Staubli VAL3: Apilar.pjx

--- Apilar.pjx ---
Parameters version=s7.10 stackSize=5000 millimeterUnit=true
Program file=_GLOBAL.pgx
Program file=_INFO.pgx
Program file=ajustar.pgx
Program file=getNum.pgx
Program file=inicializar.pgx
Program file=lower.pgx
Program file=mcp.pgx
Program file=putButton.pgx
Program file=putEx.pgx
Program file=putEx2.pgx
Program file=robot.pgx
Program file=robotGet.pgx
Program file=robotPut.pgx
Program file=start.pgx
Program file=stop.pgx
Data file=Apilar.dtx

--- Apilar.dtx ---
bool bTraslada = true
bool bFin
bool bPiezaPreparada
bool bTermina
frame fTrabajo = {x=-400, y=175, z=-274.326706, fatherId=world[0]}
jointRx jHome
public mdesc mNomSpeed = {leave=25, reach=25}
mdesc mVelAprox = {accel=25, vel=50, decel=25, blend=off}
num nPiezaActual = 1
num nTrasladadas = 7
num nPiezaAltura = 12
num nSeparacion = 100
num nTotalPiezas = 2
pointRx p0 = {ry=180, fatherId=fTrabajo[0]}
pointRx pCentro = {x=-400, y=175, z=-272, ry=180, shoulder=righty, elbow=enegative, wrist=wnegative, fatherId=world[0]}
pointRx pDestino = {x=-2.694223E-15, y=50, z=22, rx=-180, ry=7.016709E-15, rz=-180, fatherId=fTrabajo[0]}
pointRx pEntrada = {y=-50, z=103, rx=-180, rz=-180, fatherId=fTrabajo[0]}
pointRx pOrigen = {x=-1.347111E-15, y=-50, z=11, rx=-180, ry=7.016709E-15, rz=-180, fatherId=fTrabajo[0]}
pointRx pEspera = {x=-6.123234E-15, z=50, rx=-180, ry=7.016709E-15, rz=-180, fatherId=fTrabajo[0]}
pointRx pSalida = {x=-1.347111E-15, y=50, z=11, rx=-180, ry=7.016709E-15, rz=-180, fatherId=fTrabajo[0]}
tool tEyector = {z=22, fatherId=flange[0], ioLink=valve1, ioOpen=1, ioClose=1}
trsf trAprox = {z=-50}
num nEspera
num nOffset
bool bHaciaSalida
pointRx pInicio = {fatherId=world[0]}

--- start.pgx ---
program start()
begin
  // Se pone en marcha la aplicacion

  // Se inicializar la aplicacion
  call inicializar()
  call ajustar()

  // Se crean las tareas de la aplicacion
  taskCreate "mcp",100,mcp()
  taskCreate "robot",100,robot()
end

--- _GLOBAL.pgx ---
program _GLOBAL()
begin
  // BOOL
  // - bFin: indicador de finalizacion
  // - bHaciaSalida: indica la direccion del traslado de piezas
  // - bPiezaPreparada: pieza preparada para ser cogida
  // - bTermina: orden de abandonar la ejecucion de la aplicacion
  // - bTraslada: orden de trasladar la pila de piezas
  //
  // FRAME
  // frTrabajo: sistema de coordenadas del area de trabajo
  //
  // JOINT
  // - jHome: brazo en la posicion de referencia
  //
  // MDESC
  // - mNomSpeed: descriptor de movimiento a velocidad nominal
  // - mVelAprox: descriptor de movimiento a velocidad de aproximacion
  //
  // NUM
  // - nEspera: tiempo de espera en la posicion de espera antes de volver a
  //   trasladar la pila de piezas
  // - nOffset: desplazamiento de la posicion de reposo con respecto a la
  //   altura de la pila de piezas.
  // - nPiezaActual: posicion de la proxima pieza a trasladar en la pila origen
  // - nPiezaAltura: altura de la pieza a trasladar
  // - nSeparacion: distancia entre las pilas de bloques
  // - nTotalPiezas: numero total de piezas en la pila
  // - nTrasladadas: numero total acumulado de piezas trasladadas
  //
  // POINT
  // - p0: punto situado en el centro de coordenadas del espacio de trabajo
  // - pCentro: posicion central de referencia del espacio de trabajo
  // - pDestino: posicion de la proxima pieza a colocar
  // - pEntrada: posicion de la pila de entrada
  // - pEspera: posicion de reposo
  // - pInicio: posicion inicial que señala la posicion de la pila de entrada
  // - pOrigen: posicion de la proxima pieza a coger
  // - pSalida: posicion de la pila de salida
  //
  // TOOL
  // - tEyector: parametros de la herramienta (eyector de vacio con ventosas)
  //
  // TRSF
  // - trAprox: transformacion de aproximacion a las posiciones origen/destino
end

--- _INFO.pgx ---
program _INFO()
begin
  // APLILAR (Nivel 2)
  //
  // Traslada indefinidamente una pila de un determinado numero de piezas de
  // una posicion a otra.
  //
  // Version 0.0
  // copyright (c) 2022 victortorreslopez
  // GNU General Public License
  //
  // HISTORIAL DE VERSIONES
  // ----------------------
  // 0.0, 13/12/2022, VTL: creacion (desde PickPlace, 2018)
  //
  // FUNCIONALIDAD
  // -------------
  // - F1: Activa/Desactiva el modo "Trasladar".
  // - F3: Edita el numero total de piezas en la pila a trasladar.
  // - F4: Ajusta el tiempo de espera entre traslados.
  // - F6: Reinicia el contador total de piezas trasladadas.
  // - F8: Sale de la aplicacion.
  //
  // SITUACION INICIAL
  // -----------------
  // - Brazo en su posicion de referencia.
  // - Pila con el numero determinado de bloques en la posicion de entrada.
  // - Ninguna pieza en la posicion de salida.
  // - Antes de ejecutar por primera vez la aplicacion deben ajustarse al valor
  //   deseado las variables: nEspera, nPiezaAltura y nSeparacion.
  //
  // RECURSOS
  // --------
  // - Datos: BOOL, FRAME, JOINT, MDESC, POINT, STRING, TOOL, TRSF.
  // - Instrucciones: appro, title, userPage, while, cls, call, toString, if,
  //   getKey, switch, delay, movej, waitEndMove, for, taskCreate.
  // - Funciones:  getNum, lower, putButton, putEx, putEx2, robotGet, robotPut
  //
  // NOTAS
  // -----
  // - El area de trabajo es una plataforma elevada a 100 mm del suelo.
  // - Pilas de entrada y salida simetricas con respecto al centro del espacio
  //   de trabajo a una distancia "nSeparacion".
  // - En el modo trasladar las piezas se trasladan indefinidamente de la pila
  //   de entrada a la de salida y viceversa.
  // - El espacio de trabajo (fTrabajo) se determina a partir de una posicion
  //   que determina su centro de coordenadas (pCentro)
  //
  // REFERENCIAS
  // -----------
  //
  // CELDA
  // -----
  // - Version: s7.10
  // - Tipo de robot: TX60
  // - Montaje: suelo
  // - Modo usrIn0: directo.
  //
  // DATOS
  // -----
  // - Plataforma = 400x300x3 mm
  // - Altura de la plataforma = 100 mm
  // - Pieza = 69x23x12 mm
  // - Herramienta (eyector) = 40.0x33.3x22.0 mm
end

--- ajustar.pgx ---
program ajustar()
begin
  // Calcula la posiciones de referencia

  // Posicion de entrada y salida
  // - Simetricas con respecto al origen (nSeparacion)
  // - A la altura de la primera pieza
  pEntrada=appro(p0,{0,-nSeparacion/2,-nPiezaAltura,0,0,0})
  pSalida=appro(p0,{0,nSeparacion/2,-nPiezaAltura,0,0,0})

  // Posicion de espera en el centro por encima (offset) de la altura de la pila
  pEspera=appro(p0,{0,0,-((nTotalPiezas*nPiezaAltura)+nOffset),0,0,0})

  // Posicion de espera inicial por encima (offset) de la pila de entrada
  pInicio=appro(pEntrada,{0,0, -((nTotalPiezas*nPiezaAltura)+nOffset),0,0,0})
  end

--- getNum.pgx ---
public program getNum(num nX, num nY, string sFormat, num& nValue)
  local num i
  local num n
  local string s
begin
  // Acquires a number
  //
  // copyright (c) 2013-2021 victortorreslopez
  //
  // GNU General Public License
  //
  // Parameters
  // - nX: cursor column (0 to 39)
  // - nY: cursor row (0 to 13)
  // - sFormat: display format
  // - &nValue: numerical variable to be set
  //
  // Local variables
  // - i: iterator index
  // - n: number of characters in nValue
  // - s: a string
  //
  // Version history
  // ---------------
  // 0.1, 2021/12/30, VTL: 1s update (coding style)
  // 0.0, 2013/12/10, VTL: alfa release

  // Fills s with spaces
  s = ""
  n = len(toString(sFormat, nValue))
  for i = 0 to n - 1
    s = s + " "
  endFor

  // Displays spaces before acquires the new string value
  gotoxy(nX, nY)
  put(s)

  // Acquires the new numerical value
  gotoxy(nX, nY)
  get(nValue)
end

--- inicializar.pgx ---
program inicializar()
begin
  // Pone en marcha la aplicacion

  // Se establece el valor inicial de variables globales
  // BOOL
  bFin=false
  bHaciaSalida=true
  bPiezaPreparada=false
  bTermina=false
  bTraslada=false

  // FRAME
  // Se determina el centro de coordenadas de fTrabajo a partir de la posicion
  // central de referencia de todo el espacio de trabajo (pCentro)
  fTrabajo.trsf.x=pCentro.trsf.x
  fTrabajo.trsf.y=pCentro.trsf.y
  fTrabajo.trsf.z=pCentro.trsf.z

  // NUM
  nOffset=5
  nPiezaActual=0
  nPiezaAltura=12
  nSeparacion=100
  nTotalPiezas=1
  nTrasladadas=0
end

--- lower.pgx ---
public program lower(string& sText)
  local num i
  local num n
begin
  // Converts all lowercase letter of a string to uppercase
  //
  // copyright (c) 2017-2021 victortorreslopez
  //
  // GNU General Public License
  //
  // Parameters
  // - &sText: source string
  //
  // Local variables
  // - i: iterator index
  // - n: current char unicode code
  //
  // Version history
  // ---------------
  // 0.0, 2021/12/21, VTL: 1st update (coding style)
  // 0.0, 2017/01/04, VTL: alfa release

  for i = 0 to len(sText) - 1
    n = asc(sText, i)
    if (n > 65) and (n < 90)
      sText = replace(sText, chr(n + 32), 1, i)
    endIf
  endFor
end

--- mcp.pgx ---
program mcp()
  local num nTecla
begin
  // Controla la pantalla del mando manual (MCP)
  //
  // Variables locales
  // - nTecla: codigo de la tecla pulsada

  // Se establece el titulo de la aplicacion
  title("APILAR")

  // Se establece la pagina de usuario en la pantalla
  userPage()

  // Bucle principal de la tarea
  while !bFin
    // Se borra la pantalla
    cls()

    // Se muestra informacion en la pantalla
    call putEx(2,2,"Total       = "+toString("4",nTotalPiezas))
    call putEx(2,3,"Maniobras   = "+toString("4",nTrasladadas))
    call putEx(2,4,"Tpo. Espera = "+toString("4",nEspera))

    if bHaciaSalida
      call putEx2("center",8,"Entrada = "+toString("0",nTotalPiezas-nPiezaActual)+" -> "+toString("0",nPiezaActual)+" = Salida")
    else
      call putEx2("center",8,"Entrada = "+toString("0",nPiezaActual)+" <- "+toString("0",nTotalPiezas-nPiezaActual)+" = Salida")
    endIf

    // Se muestran las etiquetas de las teclas de funcion
    if bTraslada
      call putButton(1,"Para")
    else
      call putButton(3,"Total")
      call putButton(1,"Traslada")
    endIf
    call putButton(4,"Espera")
    call putButton(6,"Reset")
    call putButton(8,"Salir")

    // Se procesa la tecla pulsada
    nTecla=getKey()
    switch nTecla
      // Enter - Orden de continuar
      case 270
        bPiezaPreparada=true
      break
      // F1 - Conmuta el modo "Trasladar"
      case 271
        bTraslada=!bTraslada
      break
      // F3 - Orden de editar el numero de piezas a trasladar
      case 273
        // Se ignora mientras se trasladan piezas
        if !bTraslada
          call getNum(19,2,"4",nTotalPiezas)
          call ajustar()
        endIf
      break
      // F4 - Ajusta el tiempo de espera entre traslados
      case 274
        call getNum(19,4,"4",nEspera)
      break
      // F6 - Orden de reinicar el contador de maniobras
      case 276
        nTrasladadas=0
      break
      // F8 - Orden de salir de la aplicacion
      case 278
        bTermina=true
      break
    endSwitch

    // Se da paso a la siguiente tarea y se estabiliza la pantalla
    delay(0.1)
  endWhile
  bFin=false

  // Se muestra un mensaje de despedida
  cls()
  call putEx2("center",7,"That's all folks")
end

--- putButton.pgx ---
public program putButton(num nValue, string sText)
begin
  // Puts a text label above a function key
  //
  // Labels greater than 4 characters will shorten to 4
  //
  // copyright (c) 2015-2021 victortorreslopez
  //
  // GNU General Public License
  //
  // Parameters
  // - nValue: number of function key (1..8)
  // - sText: function key label
  //
  // References
  // - "2005-27 Example Application". Staubli. 2005
  //
  // Version history
  // ---------------
  // 0.1, 2021/12/21, VTL: centers the label
  // 0.0, 2015/01/14, VTL: alfa release

  if (nValue >= 1) and (nValue <= 8)
    if (len(sText) > 4)
      sText = left(sText, 3) + "."
    endIf
    gotoxy(((nValue - 1) * 5) + round((5 - len(sText)) / 2), 13)
    put(sText)
  endIf
end

--- putEx.pgx ---
public program putEx(num nX, num nY, string sText)
begin
  // Displays a text at the cursor position (x,y)
  //
  // The cursor is positioned on the character after the last character of
  // the message displayed
  //
  // copyright (c) 2015-2018 victortorreslopez
  //
  // GNU General Public License
  //
  // Parameters
  // - nX: cursor column (0 to 39)
  // - nY: cursor row (0 to 13)
  // - sText: character string type expression
  //
  // Version history
  // ---------------
  // 2.0, 2020/02/15, VTL: renames all parameters
  // 1.0, 2018/09/28, VTL: renames "sText" by "s"
  // 0.0, 2015/01/15, VTL: alfa release

  gotoxy(nX, nY)
  put(sText)
end

--- putEx2.pgx ---
public program putEx2(string sX, num nY, string sText)
  local num nX
begin
  // Displays a text at [left/center/right] horizontal position
  //
  // The cursor is positioned on the character after the last character of
  // the message displayed
  //
  // copyright (c) 2020 victortorreslopez
  //
  // GNU General Public License
  //
  // Parameters
  // - sX: horizontal alignment (left, center, right)
  // - nY: cursor row (0 to 13)
  // - sText: character string type expression
  //
  // Locals variables
  // - nX: cursor column (0 to 39)
  //
  // Version history
  // ---------------
  // 0.0, 2020/11/21, VTL: alfa release from "_put"

  call lower(sX)

  if len(sText) > 40
    nX = 0
  else
    if sX == "right"
      nX = 40 - len(sText)
    elseIf sX == "center"
      nX = (40 - len(sText)) / 2
    elseIf sX == "left"
      nX = 0
    endIf
  endIf

  gotoxy(nX, nY)
  put(sText)
end

--- robot.pgx ---
program robot()
begin
  // Controla los movimientos del brazo

  // Se desplaza a la posicion de reposo
  movej(pInicio,tEyector,mNomSpeed)
  waitEndMove()

  // Bucle principal de la tarea
  while !bTermina
    if bTraslada
      // Traslada las piezas desde la entrada a la salida
      bHaciaSalida=true
      for nPiezaActual=0 to nTotalPiezas-1
        // Calcula la posicion de la proxima pieza a coger
        pOrigen=appro(pEntrada,{0,0,-(nTotalPiezas-1-nPiezaActual)*nPiezaAltura,0,0,0})
        // Calcula la posicion de la proxima pieza a colocar
        pDestino=appro(pSalida,{0,0,-nPiezaActual*nPiezaAltura,0,0,0})

        // Se coge una pieza
        call robotGet(pOrigen,trAprox,tEyector,mNomSpeed,mVelAprox)
        // Se coloca una pieza
        call robotPut(pDestino,trAprox,tEyector,mNomSpeed,mVelAprox)

        // Se actualiza el contador de maniobras
        nTrasladadas=nTrasladadas+1
      endFor

      // Se regresa a la posicion de reposo
      movej(pEspera,tEyector,mNomSpeed)
      waitEndMove()
      delay(nEspera)

      // Traslada las piezas desde la salida a la entrada
      bHaciaSalida=false
      for nPiezaActual=0 to nTotalPiezas-1
        // Calcula la posicion de la proxima pieza a coger
        pOrigen=appro(pSalida,{0,0,-(nTotalPiezas-1-nPiezaActual)*nPiezaAltura,0,0,0})
        // Calcula la posicion de la proxima pieza a colocar
        pDestino=appro(pEntrada,{0,0,-nPiezaActual*nPiezaAltura,0,0,0})

        // Se coge una pieza
        call robotGet(pOrigen,trAprox,tEyector,mNomSpeed,mVelAprox)
        // Se coloca una pieza
        call robotPut(pDestino,trAprox,tEyector,mNomSpeed,mVelAprox)

        // Se actualiza el contador de maniobras
        nTrasladadas=nTrasladadas+1
      endFor

      // Se regresa a la posicion de reposo
      movej(pEspera,tEyector,mNomSpeed)
      waitEndMove()
      delay(nEspera)
    endIf

    // Se situa sobre la pila de entrada
    movej(pInicio,tEyector,mNomSpeed)
    waitEndMove()

    // Se da paso a la siguiente tarea
    delay(0)
  endWhile
  bTermina=false

  // Se regresa a la posicion de referencia
  movej(jHome,tEyector,mNomSpeed)
  waitEndMove()

  // Se informa de la finalizacion de la tarea
  bFin=true
end

--- robotGet.pgx ---
public program robotGet(point pPosition, trsf trTrans, tool tTool, mdesc mApproach, mdesc mTarget)
  local point pAppro
begin
  // Picks a part
  //
  // copyright (c) 2015-2018 victortorreslopez
  //
  // GNU General Public License
  //
  // Parameters
  // - pPosition: target position
  // - trTrans: approach transform to target position
  // - tTool: current tool
  // - mApproach: movement descriptor to "approach" point
  // - mTarget: movement descriptor to "target" position
  //
  // Local variables
  // - pAppro: approach point to target position
  //
  // References
  // - "2005-27 Example Application". Staubli. 2005
  //
  // Version history
  // ---------------
  // 2.0, 2020/02/15, VTL: renames all parameters
  // 1.1, 2018/09/27, VTL: adds "ma"
  // 1.0, 2018/09/27, VTL: renames "m" by "mt"
  // 0.0, 2015/01/14, VTL: alfa release

  pAppro = appro(pPosition, trTrans)
  movej(pAppro, tTool, mApproach)
  movel(pPosition, tTool, mTarget)
  close(tTool)
  movel(pAppro, tTool, mTarget)
end

--- robotPut.pgx ---
public program robotPut(point pPosition, trsf trTrans, tool tTool, mdesc mApproach, mdesc mTarget)
  local point pAppro
begin
  // Places a part
  //
  // copyright (c) 2015 victortorreslopez
  //
  // GNU General Public License
  //
  // Parmeters
  // - pPosition: target position
  // - trTrans: approach transform to target position
  // - tTool: tool
  // - mApproach: movement descriptor to "approach" point
  // - mTarget: movement descriptor to "target" position
  //
  // Local variables
  // - pAppro: approach point to target position
  //
  // References
  // - "2005-27 Example Application". Staubli. 2005
  //
  // Version history
  // ---------------
  // 2.0, 2020/02/15, VTL: renames all parameters
  // 1.1, 2018/09/27, VTL: add "ma"
  // 1.0, 2018/09/27, VTL: rename "m" by "mt"
  // 0.0, 2015/01/14, VTL: alfa release
  //
  pAppro = appro(pPosition, trTrans)
  movej(pAppro, tTool, mApproach)
  movel(pPosition, tTool, mTarget)
  open(tTool)
  movel(pAppro, tTool, mTarget)
end
